RoboDK station: Station TEST (1).rdk

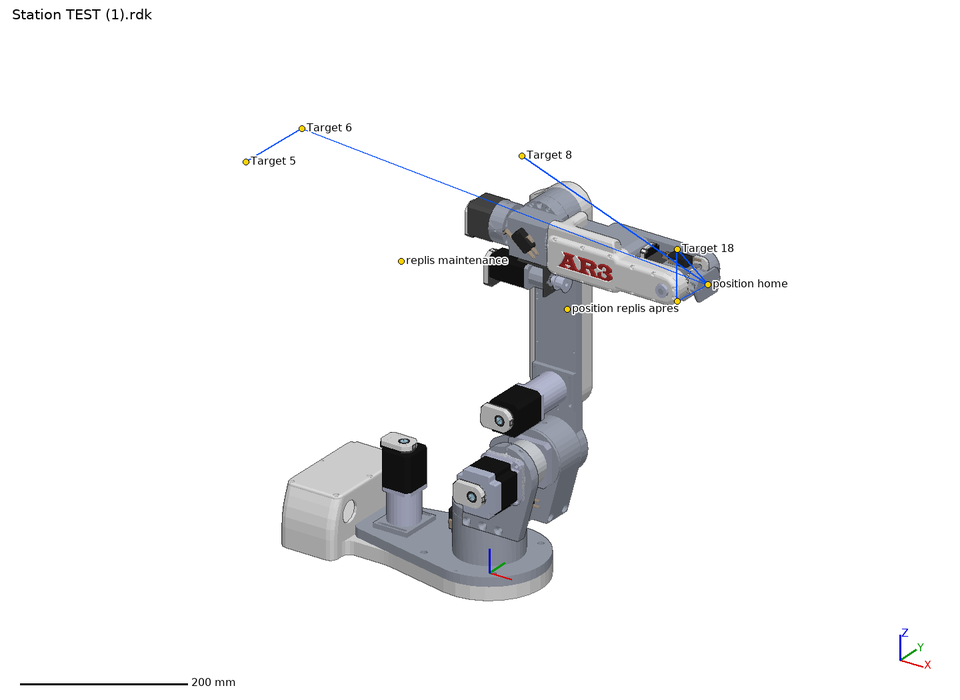
[picture v0: the station drawn from its stored meshes, robots at their saved joint values, targets as dots, program paths as lines]
Station Station TEST (1) (saved by RoboDK 5.6.3). Poses are relative to the parent item; angles as X-Y-Z fixed-axis rotations.
  - frame Annin Robotics AR3 Base at (0, 0, 0) mm
    - robot Annin Robotics AR3: 6 axes
        modified DH rows (alpha deg, a mm, theta deg, d mm): 0, 0, 0, 169.78; -90, 64.15, 0, -6.99; 0, 305, -90, 0; -90, 0, 0, 222.94; 90, 0, 0, 0; -90, 0, 180, 35.9
        joint limits [-170, -132, 1, -165, -105, -155] to [170, 0, 141, 165, 105, 155]; home [0, -90, 90, 0, 0, 0]; saved at [0, -90, 90, 0, 0, 0]
    - target position replis apres defaut (Cartesian target) at (118.65, -6.99, 385.01) mm, rotated rx -180 ry 87.47 rz -180 deg; joints [0, -132, 134.53, 0, 0, 0] of Annin Robotics AR3
    - target position home (Cartesian target) at (322.99, -6.99, 474.78) mm, rotated rx 0 ry 90 rz 0 deg; joints [0, -90, 90, 0, 0, 0] of Annin Robotics AR3
    - target replis maintenance (Cartesian target) at (-118.06, -13.72, 385.01) mm, rotated rx -180 ry 87.47 rz 10 deg; joints [170, -132, 134.53, 0, 0, 0] of Annin Robotics AR3
    - target Target 5 (Cartesian target) at (-319.3, -49.2, 474.83) mm, rotated rx 0 ry 89.99 rz -170 deg; joints [170, -90, 89.99, 0, 0, 0] of Annin Robotics AR3
    - target Target 6 (Cartesian target) at (-316.87, 62.97, 474.83) mm, rotated rx 0 ry 89.99 rz 170 deg; joints [-170, -90, 89.99, 0, 0, 0] of Annin Robotics AR3
    - target Target 6 (Cartesian target) at (-316.87, 62.97, 474.83) mm, rotated rx 0 ry 89.99 rz 170 deg; joints [-170, -90, 89.99, 0, 0, 0] of Annin Robotics AR3
    - target Target 7 (Cartesian target) at (322.99, -6.99, 474.83) mm, rotated rx 0 ry 89.99 rz 0 deg; joints [0, -90, 89.99, 0, 0, 0] of Annin Robotics AR3
    - target Target 8 (Cartesian target) at (52.39, -6.99, 569.67) mm, rotated rx 0 ry 47.99 rz 0 deg; joints [0, -132, 89.99, 0, 0, 0] of Annin Robotics AR3
    - target Target 9 (Cartesian target) at (52.39, -6.99, 569.67) mm, rotated rx 0 ry 47.99 rz 0 deg; joints [0, -132, 89.99, 0, 0, 0] of Annin Robotics AR3
    - target Target 10 (Cartesian target) at (322.99, -6.99, 474.83) mm, rotated rx 0 ry 89.99 rz 0 deg; joints [0, -90, 89.99, 0, 0, 0] of Annin Robotics AR3
    - target Target 11 (Cartesian target) at (322.99, -6.99, 474.78) mm, rotated rx -90 ry -75 rz -90 deg; joints [0, -90, 90, -165, 0, 0] of Annin Robotics AR3
    - target Target 12 (Cartesian target) at (322.99, -6.99, 474.78) mm, rotated rx -90 ry -75 rz -90 deg; joints [0, -90, 90, -165, 0, 0] of Annin Robotics AR3
    - target Target 13 (Cartesian target) at (322.99, -6.99, 474.78) mm, rotated rx 90 ry -75 rz 90 deg; joints [0, -90, 90, 165, 0, 0] of Annin Robotics AR3
    - target Target 14 (Cartesian target) at (322.99, -6.99, 474.78) mm, rotated rx 90 ry -75 rz 90 deg; joints [0, -90, 90, 165, 0, 0] of Annin Robotics AR3
    - target Target 15 (Cartesian target) at (322.99, -6.99, 474.78) mm, rotated rx 0 ry 90 rz 0 deg; joints [0, -90, 90, 0, 0, 0] of Annin Robotics AR3
    - target Target 16 (Cartesian target) at (322.99, -6.99, 474.78) mm, rotated rx 0 ry 90 rz 0 deg; joints [0, -90, 90, 0, 0, 0] of Annin Robotics AR3
    - target Target 17 (Cartesian target) at (277.8, -6.99, 440.1) mm, rotated rx 180 ry -15 rz -180 deg; joints [0, -90, 90, 0, -105, 0] of Annin Robotics AR3
    - target Target 18 (Cartesian target) at (277.8, -6.99, 509.46) mm, rotated rx 0 ry -15 rz 0 deg; joints [0, -90, 90, 0, 105, 0] of Annin Robotics AR3
    - target Target 19 (Cartesian target) at (322.99, -6.99, 474.78) mm, rotated rx 0 ry 90 rz 0 deg; joints [0, -90, 90, 0, 0, 0] of Annin Robotics AR3
    - target Target 20 (Cartesian target) at (322.99, -6.99, 474.78) mm, rotated rx 0 ry 90 rz 0 deg; joints [0, -90, 90, 0, 0, 0] of Annin Robotics AR3
    - target Target 21 (Cartesian target) at (322.99, -6.99, 474.78) mm, rotated rx -90 ry -65 rz -90 deg; joints [0, -90, 90, 0, 0, -155] of Annin Robotics AR3
    - target Target 22 (Cartesian target) at (322.99, -6.99, 474.78) mm, rotated rx 0 ry 90 rz 0 deg; joints [0, -90, 90, 0, 0, 0] of Annin Robotics AR3
    - target Target 23 (Cartesian target) at (322.99, -6.99, 474.78) mm, rotated rx 0 ry 90 rz 0 deg; joints [0, -90, 90, 0, 0, 0] of Annin Robotics AR3
    - target Target 24 (Cartesian target) at (322.99, -6.99, 474.78) mm, rotated rx 0 ry 90 rz 0 deg; joints [0, -90, 90, 0, 0, 0] of Annin Robotics AR3
    - target Target 25 (Cartesian target) at (322.99, -6.99, 474.78) mm, rotated rx 90 ry -64 rz 90 deg; joints [0, -90, 90, 0, 0, 154] of Annin Robotics AR3
    - target Target 26 (Cartesian target) at (322.99, -6.99, 474.78) mm, rotated rx 0 ry 90 rz 0 deg; joints [0, -90, 90, 0, 0, 0] of Annin Robotics AR3
    - target Target 27 (Cartesian target) at (322.99, -6.99, 474.78) mm, rotated rx 0 ry 90 rz 0 deg; joints [0, -90, 90, 0, 0, 0] of Annin Robotics AR3
  - program replis apres defaut (2 instructions, listed below)
  - program replis maintenance (2 instructions, listed below)
  - program position home (2 instructions, listed below)
  - program verification axe (17 instructions, listed below)
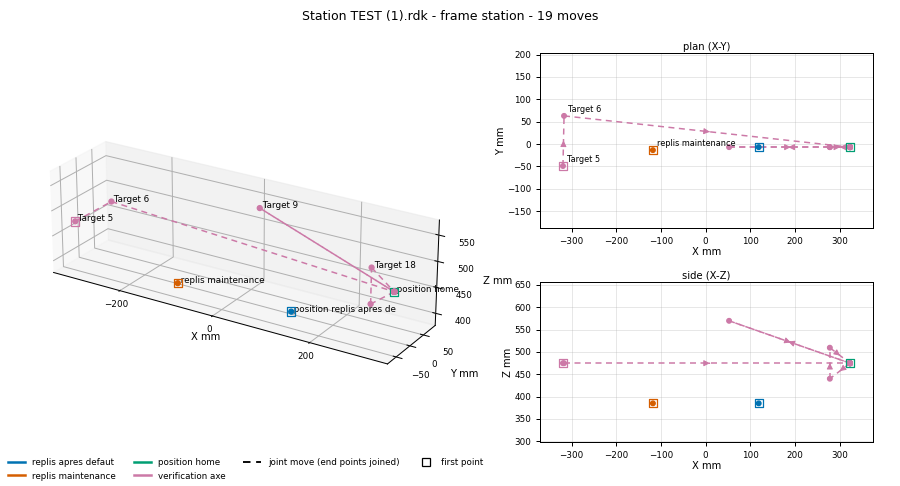
[picture p0: tool path of Station TEST (1).rdk in frame station, 19 of 19 moves have a stored position in this frame; points joined in program order, loops and branches not executed]

--- program replis apres defaut (robot Annin Robotics AR3) ---
  Définir Ref.: Annin Robotics AR3 Base
  MoveJ (position replis apres defaut)

--- program replis maintenance (robot Annin Robotics AR3) ---
  Définir Ref.: Annin Robotics AR3 Base
  MoveJ (replis maintenance)

--- program position home (robot Annin Robotics AR3) ---
  Définir Ref.: Annin Robotics AR3 Base
  MoveJ (position home)

--- program verification axe (robot Annin Robotics AR3) ---
  Définir Ref.: Annin Robotics AR3 Base
  MoveJ (Target 5)
  MoveJ (Target 6)
  MoveJ (Target 7)
  MoveJ (Target 9)
  MoveJ (Target 10)
  MoveJ (Target 12)
  MoveJ (Target 14)
  MoveJ (Target 15)
  MoveJ (Target 17)
  MoveJ (Target 18)
  MoveJ (Target 19)
  MoveJ (Target 21)
  MoveJ (Target 21)
  MoveJ (Target 23)
  MoveJ (Target 25)
  MoveJ (Target 27)
